// Mitsubishi GX Works2 project: 타이머 점멸 예제 1   PLC: Q03UDV

PROGRAM MAIN
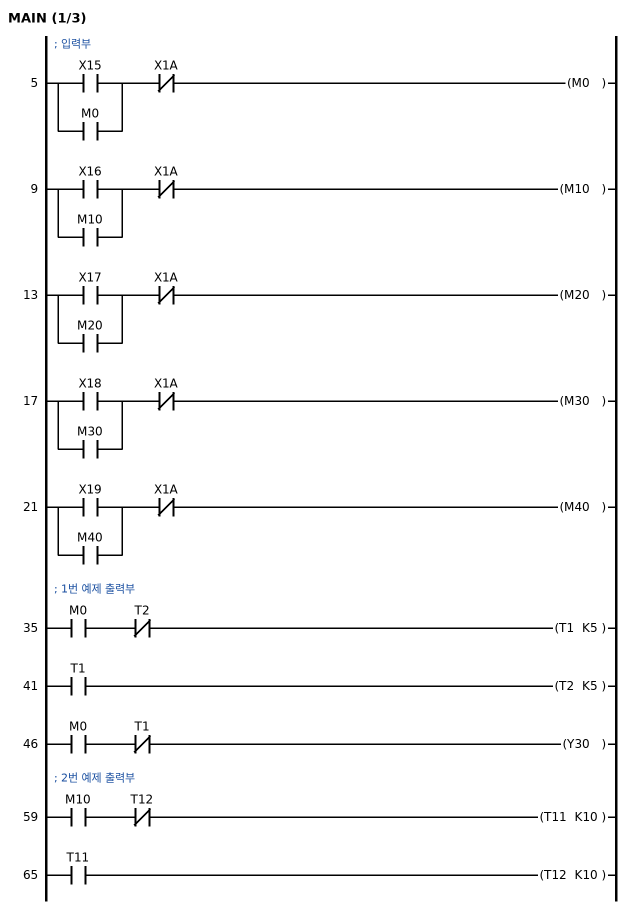
; 입력부
5     LD      X15
      OR      M0
      ANI     X1A
      OUT     M0
9     LD      X16
      OR      M10
      ANI     X1A
      OUT     M10
13    LD      X17
      OR      M20
      ANI     X1A
      OUT     M20
17    LD      X18
      OR      M30
      ANI     X1A
      OUT     M30
21    LD      X19
      OR      M40
      ANI     X1A
      OUT     M40
; 1번 예제 출력부
35    LD      M0
      ANI     T2
      OUT     T1 K5
41    LD      T1
      OUT     T2 K5
46    LD      M0
      ANI     T1
      OUT     Y30
; 2번 예제 출력부
59    LD      M10
      ANI     T12
      OUT     T11 K10
65    LD      T11
      OUT     T12 K10
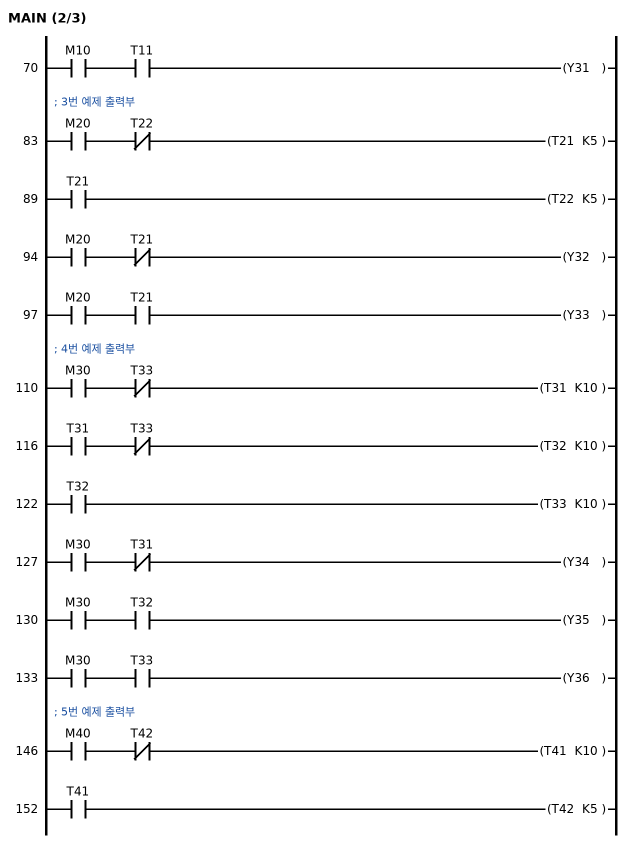
70    LD      M10
      AND     T11
      OUT     Y31
; 3번 예제 출력부
83    LD      M20
      ANI     T22
      OUT     T21 K5
89    LD      T21
      OUT     T22 K5
94    LD      M20
      ANI     T21
      OUT     Y32
97    LD      M20
      AND     T21
      OUT     Y33
; 4번 예제 출력부
110   LD      M30
      ANI     T33
      OUT     T31 K10
116   LD      T31
      ANI     T33
      OUT     T32 K10
122   LD      T32
      OUT     T33 K10
127   LD      M30
      ANI     T31
      OUT     Y34
130   LD      M30
      AND     T32
      OUT     Y35
133   LD      M30
      AND     T33
      OUT     Y36
; 5번 예제 출력부
146   LD      M40
      ANI     T42
      OUT     T41 K10
152   LD      T41
      OUT     T42 K5
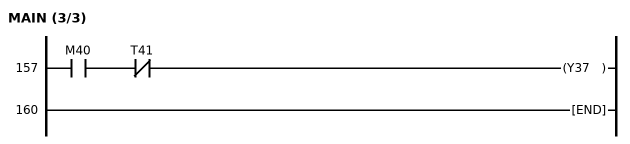
157   LD      M40
      ANI     T41
      OUT     Y37
160   END
END_PROGRAM
